FUNCTION_BLOCK ZeroLimitsTest EXTENDS TcUnit_Zeugwerk.FB_TestSuite

Test_PositionInterface();
Test_PositionInterfaceValidateInput();
Test_PositionInterfaceValidateInput_1();
Test_VelocityInterface();
Test_VelocityInterface_1();
Test_VelocityInterfaceValidateInput();

METHOD Test_PositionInterface
VAR_INST
  otg : Struckig.Otg(0.005, 3) := (
    CurrentPosition :=     [ 0.0, -2.0, 0.0 ],
    CurrentVelocity :=     [ 0.2, 0.0, 0.0 ],
    CurrentAcceleration := [ 0.0, 0.0, 0.0 ],
    TargetPosition :=      [ 1.0, -3.0, 0.0 ],
    TargetVelocity :=      [ 0.2, 0.0, 0.0 ],
    TargetAcceleration :=  [ 0.0, 0.0, 0.0 ],
    MaxVelocity :=         [ 1.0, 1.0, 1.0 ],
    MaxAcceleration :=     [ 0.0, 1.0, 0.0 ],
    MaxJerk :=             [ 0.0, 1.0, 0.0 ]
  );
END_VAR
TEST('Test_PositionInterface');

otg();
AssertEquals_INT(otg.State, Struckig.TrajectoryState.Busy, message:='Trajectory working');
AssertEquals_LREAL(5.0, otg.Duration, 1E-6, message:='Duration not met');


TEST_FINISHED();
END_METHOD

METHOD Test_PositionInterfaceValidateInput
VAR_INST
  otg : Struckig.Otg(0.005, 3) := (
    CurrentPosition :=     [ 0.0, -2.0, 0.0 ],
    CurrentVelocity :=     [ -0.2, 0.0, 0.0 ],
    CurrentAcceleration := [ 1.0, 0.0, 0.0 ],
    TargetPosition :=      [ 0.4, -3.0, 0.0 ],
    TargetVelocity :=      [ 0.8, 0.0, 0.0 ],
    TargetAcceleration :=  [ 1.0, 0.0, 0.0 ],
    MaxVelocity :=         [ 1.0, 200.0, 1.0 ],
    MaxAcceleration :=     [ 1.0, 200.0, 0.0 ],
    MaxJerk :=             [ 0.0, 200.0, 0.0 ]
  );
END_VAR
TEST('Test_PositionInterfaceValidateInput');

otg();
AssertEquals_INT(Struckig.TrajectoryState.Error, otg.State, message:='Trajectory failed');
AssertEquals_STRING('Zero limits conflict in step 1', otg.ErrorMessage(), message:='');


TEST_FINISHED();
END_METHOD

METHOD Test_PositionInterfaceValidateInput_1
VAR_INST
  otg : Struckig.Otg(0.005, 3) := (
    CurrentPosition :=     [ 0.0, -2.0, 0.0 ],
    CurrentVelocity :=     [ -0.2, 0.0, 0.0 ],
    CurrentAcceleration := [ 1.0, 0.0, 0.0 ],
    TargetPosition :=      [ 0.3, -3.0, 0.0 ],
    TargetVelocity :=      [ 0.8, 0.0, 0.0 ],
    TargetAcceleration :=  [ 1.0, 0.0, 0.0 ],
    MaxVelocity :=         [ 1.0, 2.0, 1.0 ],
    MaxAcceleration :=     [ 1.0, 2.0, 0.0 ],
    MaxJerk :=             [ 0.0, 2.0, 0.0 ]
  );
END_VAR
TEST('Test_PositionInterfaceValidateInput_1');

otg();
AssertEquals_INT(Struckig.TrajectoryState.Error, otg.State, message:='Trajectory failed');
AssertEquals_STRING('Zero limits conflict with other degrees of freedom in time synchronization', otg.ErrorMessage(), message:='');


TEST_FINISHED();
END_METHOD

METHOD Test_VelocityInterface
VAR_INST
  otg : Struckig.Otg(0.005, 3) := (
    ControlInterface := Struckig.ControlInterfaceType.Velocity,
    CurrentPosition :=     [ 0.0, -2.0, 0.0 ],
    CurrentVelocity :=     [ -0.2, 0.0, 0.0 ],
    CurrentAcceleration := [ 1.0, 0.0, 0.2 ],
    TargetPosition :=      [ 0.4, -3.0, 0.0 ],
    TargetVelocity :=      [ 0.9, 0.5, 0.4 ],
    TargetAcceleration :=  [ 1.0, 0.0, 0.2 ],
    MaxVelocity :=         [ 1.0, 2.0, 1.0 ],
    MaxAcceleration :=     [ 1.0, 2.0, 6.0 ],
    MaxJerk :=             [ 1.0, 2.0, 0.0 ]
  );
END_VAR
TEST('Test_VelocityInterface');

otg();
AssertEquals_INT(otg.State, Struckig.TrajectoryState.Busy, message:='Trajectory working');
AssertEquals_LREAL(2.0, otg.Duration, 1E-6, message:='Duration not met');


TEST_FINISHED();
END_METHOD

METHOD Test_VelocityInterface_1
VAR_INST
  otg : Struckig.Otg(0.005, 3) := (
    ControlInterface := Struckig.ControlInterfaceType.Velocity,
    CurrentPosition :=     [ 0.0, -2.0, 0.0 ],
    CurrentVelocity :=     [ -0.2, 0.0, 0.0 ],
    CurrentAcceleration := [ 1.0, 0.0, 0.2 ],
    TargetPosition :=      [ 0.4, -3.0, 0.0 ],
    TargetVelocity :=      [ 0.9, 0.5, 0.4 ],
    TargetAcceleration :=  [ 1.0, 0.0, 0.2 ],
    MaxVelocity :=         [ 1.0, 2.0, 1.0 ],
    MaxAcceleration :=     [ 1.0, 2.0, 6.0 ],
    MaxJerk :=             [ 0.0, 2.0, 20.0 ]
  );
END_VAR
TEST('Test_VelocityInterface_1');

otg();
AssertEquals_INT(otg.State, Struckig.TrajectoryState.Busy, message:='Trajectory working');
AssertEquals_LREAL(1.1, otg.Duration, 1E-6, message:='Duration not met');


TEST_FINISHED();
END_METHOD

METHOD Test_VelocityInterfaceValidateInput
VAR_INST
  otg : Struckig.Otg(0.005, 3) := (
    ControlInterface := Struckig.ControlInterfaceType.Velocity,
    CurrentPosition :=     [ 0.0, -2.0, 0.0 ],
    CurrentVelocity :=     [ -0.2, 0.0, 0.0 ],
    CurrentAcceleration := [ 1.0, 0.0, 0.2 ],
    TargetPosition :=      [ 0.4, -3.0, 0.0 ],
    TargetVelocity :=      [ 0.9, 0.5, 0.4 ],
    TargetAcceleration :=  [ 1.0, 0.0, 0.2 ],
    MaxVelocity :=         [ 1.0, 2.0, 1.0 ],
    MaxAcceleration :=     [ 1.0, 2.0, 6.0 ],
    MaxJerk :=             [ 0.0, 2.0, 0.0 ]
  );
END_VAR
TEST('Test_VelocityInterfaceValidateInput');

otg();
AssertEquals_INT(Struckig.TrajectoryState.Error, otg.State, message:='Trajectory failed');
AssertEquals_STRING('Zero limits conflict with other degrees of freedom in time synchronization', otg.ErrorMessage(), message:='');


TEST_FINISHED();
END_METHOD

END_FUNCTION_BLOCK

(* stored: Version 1.1.0.1
   POU ZeroLimitsTest: Id {ac7f32e5-ecad-400f-91b1-3253b77ac3df}, SpecialFunc None
   Method Test_PositionInterface: Id {0829a982-07ad-4ba6-bc32-d39a377d4344}
   Method Test_PositionInterfaceValidateInput: Id {044f609b-7783-4629-890a-9966318434d9}
   Method Test_PositionInterfaceValidateInput_1: Id {d852fee9-6ec1-4b8e-92e4-d6c0dc952031}
   Method Test_VelocityInterface: Id {3edded92-d937-44ce-85aa-dd12e001375b}
   Method Test_VelocityInterface_1: Id {766c70c1-5d05-4be1-95cc-58fc2d2739c0}
   Method Test_VelocityInterfaceValidateInput: Id {4ea7e036-398c-448b-8611-436225621c2e} *)
